PROGRAM MAIN
VAR
	Temp		: LREAL;
	TempSpeed	: LREAL := 0.1;

	HeatActual	: LREAL;
	HeatSetpoint: LREAL;
	CoolActual	: LREAL;
	CoolSetpoint: LREAL;
	
	Counter	: WORD;	
	incr 	: LREAL;
	Reset		: BOOL;
END_VAR
VAR CONSTANT
	HEAT_INCR_PERSEC	: LREAL := 10;
	COOL_INCR_PERSEC	: LREAL := 3;
END_VAR

Counter := Counter + 7;

incr := HEAT_INCR_PERSEC * 1000.0 / UDINT_TO_LREAL(_TaskInfo[1].CycleTime);
HeatActual := HeatActual + SEL( HeatActual > HeatSetpoint,  incr, -incr);

incr := COOL_INCR_PERSEC * 1000.0 / UDINT_TO_LREAL(_TaskInfo[1].CycleTime);
CoolActual := CoolActual + SEL( CoolActual > CoolSetpoint,  incr, -incr);

TempSpeed := TempSpeed + 0.000007 * HeatActual - 0.000003 * CoolActual; 
Temp := Temp + TempSpeed;

IF Temp < 10 THEN
	Temp := 10;
	TempSpeed := TempSpeed / 2.0;
END_IF


IF Reset THEN
	Counter := 0;
	TempSpeed := 0;
	Temp := 0;
END_IF

END_PROGRAM

(* stored: Version 1.1.0.1, ProductVersion 3.1.4020.12
   POU MAIN: Id {9b7ef0cc-2fb3-4c0a-860d-f4f781207fb5}, SpecialFunc None *)
